    eNestState                              		:= E_NestState.IDLE;
    bSequenceToggle                         		:= FALSE; // Always restart from rotation step after reset
    GVL_MASTER.stNestTable.bNestStartCycle  		:= FALSE;
    GVL_MASTER.stNestTable.bNestInMotion    		:= FALSE;
    GVL_MASTER.stNestTable.qNestRotatePortA 		:= FALSE;
    GVL_MASTER.stNestTable.qNestRotatePortB 		:= FALSE;
    GVL_MASTER.stNestTable.bSupportExtendRequest    := FALSE;
    GVL_MASTER.stNestTable.bSupportRetractRequest   := TRUE;  // Safe home posture for elevator

    RETURN; // Abort remaining logic execution for this cycle
END_IF

// Global Safety Interlock: Force fault state immediately if air/safety is lost
IF NOT GVL_IO.stSafety.bSafetyOK AND GVL_Master.stMachineStatus.bFault THEN
    eNestState := E_NestState.FAULT;
END_IF

//eCurrentNestPos := M_GetCurrentPosition();

// =================================================================
// 2. INPUT SIGNAL PROCESSING (TRIGGERS)
// =================================================================
// Evaluate positive edge of the safety-certified two-hand control
rTrigTwoHands(CLK := GVL_IO.stSafety.bTwoHandsSafe);
tTwoHandTargetTime := REAL_TO_TIME(rHmiTwoHandPresetTime);   // Convert the HMI float milliseconds value into PLC TIME data type
tTwoHandHoldTimer(IN := GVL_IO.stSafety.bTwoHandsSafe, PT := tTwoHandTargetTime); // Execute the verification timer tied to the physical two-hand safety input

// Trigger processing to allow automated cycle start from IDLE state
// IF rTrigTwoHands.Q AND GVL_MASTER.bStations_Home AND GVL_IO.stSafety.bSafetyOK AND (eNestState = E_NestState.IDLE) THEN
//      IF GVL_MASTER.stMachineStatus.bAutoCycle THEN
//          GVL_MASTER.stNestTable.bNestInMotion := TRUE;
//          eNestState                           := E_NestState.ROTATING_TABLE; // Start the automated cycle directly at rotation step
//      END_IF
// END_IF

// =================================================================
// 3. TIMERS EXECUTION (CYCLIC COUPLING TO MAIN PROGRAM INSTANCES)
// =================================================================
// Enchained timers execution pattern to generate an automated timeline for the TESTING state
tRotatingTableDelay(IN  := (eNestState = E_NestState.ROTATING_TABLE), PT := T#500MS);
tPortB_ResetDelay(IN    := (eNestState = E_NestState.STOP_TABLE), PT := T#1S);

// TESTING TIMELINE: 
// 1. Initial 100ms settling delay starts when entering TESTING state
tSupportRetractDelay(IN := (eNestState = E_NestState.TESTING), PT := T#100MS);
// 2. 2-Second lift holding duration executes after the initial pause finishes
tSupportExtendDelay(IN  := (eNestState = E_NestState.TESTING) AND tSupportRetractDelay.Q, PT := T#200MS);

// Two-hand return timeout.
// If the operator does not press the two-hand control again within 1 second,
// the sequence goes to FAULT.
tTwoHandReturnTimeout(IN := (eNestState = E_NestState.WRONG_POSITION),PT := T#5S);

// =================================================================
// 4. NEST TABLE STATE MACHINE CONTROL (WITH INTERNAL INTERLOCKS)
// =================================================================
CASE GVL_Master.stMachineStatus.eMachineState OF    
    
    E_MachineState.SYSTEM_AUTO_CYCLE,
	E_MachineState.MANUAL_MODE:
        
        CASE eNestState OF
        
            E_NestState.IDLE:

				GVL_MASTER.stNestTable.qNestRotatePortA := FALSE;
				GVL_MASTER.stNestTable.qNestRotatePortB := FALSE;
				GVL_MASTER.stNestTable.bNestInMotion    := FALSE;
				GVL_MASTER.stProcess.bNestTestingReady  := FALSE;
			//
				IF GVL_IO.stSafety.bSafetyOK
				   AND rTrigTwoHands.Q
				   AND GVL_MASTER.bStations_Home
				   AND GVL_MASTER.stNestTable.bSupportRetracted
				   AND bNestSequenceAllowed
				   AND (
						GVL_MASTER.stMachineStatus.eMachineState =
							E_MachineState.MANUAL_MODE
						OR
						GVL_MASTER.stPuckLocker.bIndexPermissive
					)
				   AND stKistler_Status.bInPosition
				   AND NOT stKistler_Status.bBusy THEN
				
					GVL_MASTER.stNestTable.bNestInMotion := TRUE;
					eNestState := E_NestState.ROTATING_TABLE;
				
				END_IF
        
            E_NestState.ROTATING_TABLE: // State 2: ROTATING TABLE

				GVL_MASTER.stNestTable.bNestInMotion      := TRUE;
				GVL_MASTER.stProcess.bNestTestingReady    := FALSE;
				GVL_MASTER.stNestTable.bSupportExtendRequest := FALSE;
			    GVL_MASTER.stNestTable.bSupportRetractRequest := TRUE;
			
				IF NOT GVL_IO.stSafety.bSafetyOK THEN
			
					GVL_MASTER.stNestTable.qNestRotatePortA := FALSE;
					GVL_MASTER.stNestTable.qNestRotatePortB := FALSE;
					eNestState := E_NestState.FAULT;
			
				ELSIF NOT GVL_IO.stSafety.bTwoHandsSafe
					  AND NOT tTwoHandHoldTimer.Q THEN
			
					GVL_MASTER.stNestTable.qNestRotatePortA := FALSE;
					GVL_MASTER.stNestTable.qNestRotatePortB := FALSE;
					eNestState := E_NestState.WRONG_POSITION;
			
				ELSIF NOT bNestSequenceAllowed THEN
			
					GVL_MASTER.stNestTable.qNestRotatePortA := FALSE;
					GVL_MASTER.stNestTable.qNestRotatePortB := FALSE;
					eNestState := E_NestState.IDLE;
			
				ELSIF GVL_MASTER.stNestTable.bSupportRetracted 
					AND NOT stKistler_Status.bBusy 
					AND NOT GVL_MASTER.stActuators.bGuideCylinderExtendRequest
					AND stKistler_Status.bInPosition
					AND NOT GVL_MASTER.stProcess.bKistlerCycleRequest THEN
			
					GVL_MASTER.stNestTable.qNestRotatePortA := TRUE;
					GVL_MASTER.stNestTable.qNestRotatePortB := FALSE;
			
					IF tRotatingTableDelay.Q
					   AND GVL_MASTER.stNestTable.bNestCompletedSensor THEN
			
						eNestState := E_NestState.STOP_TABLE;
			
					END_IF
			
				ELSE
					// Support is not retracted. Do not rotate.
					GVL_MASTER.stNestTable.qNestRotatePortA := FALSE;
					GVL_MASTER.stNestTable.qNestRotatePortB := FALSE;
			
				END_IF
        
            E_NestState.STOP_TABLE: // State 3: STOP TABLE

				GVL_MASTER.stProcess.bNestTestingReady := FALSE;
			
				GVL_MASTER.stNestTable.qNestRotatePortA := FALSE;
				GVL_MASTER.stNestTable.qNestRotatePortB := TRUE;
			
				IF NOT GVL_IO.stSafety.bSafetyOK THEN
			
					GVL_MASTER.stNestTable.qNestRotatePortA := FALSE;
					GVL_MASTER.stNestTable.qNestRotatePortB := FALSE;
					eNestState := E_NestState.FAULT;
			
				ELSIF NOT bNestSequenceAllowed THEN
			
					GVL_MASTER.stNestTable.qNestRotatePortA := FALSE;
					GVL_MASTER.stNestTable.qNestRotatePortB := FALSE;
					GVL_MASTER.stNestTable.bNestInMotion    := FALSE;
					eNestState := E_NestState.IDLE;
			
				ELSIF tPortB_ResetDelay.Q
					  AND GVL_MASTER.stNestTable.bNestReadySensor
					  AND GVL_MASTER.stNestTable.bNestLockedSensor THEN
			
					GVL_MASTER.stNestTable.bNestInMotion    := FALSE;
					GVL_MASTER.stNestTable.qNestRotatePortB := FALSE;
					eNestState := E_NestState.TESTING;
			
				END_IF
        
			E_NestState.TESTING: // State 4: TESTING / Kistler test position
			
				GVL_MASTER.stNestTable.qNestRotatePortA := FALSE;
				GVL_MASTER.stNestTable.qNestRotatePortB := FALSE;
				GVL_MASTER.stNestTable.bNestInMotion := FALSE;
			
			
				IF NOT GVL_IO.stSafety.bSafetyOK THEN
			
					GVL_MASTER.stProcess.bNestTestingReady := FALSE;
					eNestState := E_NestState.FAULT;
			
			
				ELSIF NOT bNestSequenceAllowed THEN
			
					GVL_MASTER.stProcess.bNestTestingReady := FALSE;
					eNestState := E_NestState.IDLE;
			
			
				ELSIF NOT GVL_MASTER.stNestTable.bNestReadySensor
					  OR NOT GVL_MASTER.stNestTable.bNestLockedSensor
					  OR eCurrentNestPos = E_NestPosition.Unknown THEN
			
					GVL_MASTER.stProcess.bNestTestingReady := FALSE;
					eNestState := E_NestState.FAULT;
			
			
				ELSE
			
					// Table is stopped and safely positioned for the Kistler process.
					GVL_MASTER.stProcess.bNestTestingReady := TRUE;
			
			
					// The Process Cycle has completed the Kistler operation
					// and is requesting the nest to leave the testing phase.
					IF GVL_MASTER.stProcess.bReleaseNestRotation THEN
			
						GVL_MASTER.stProcess.bNestTestingReady := FALSE;
						GVL_MASTER.stProcess.bReleaseNestRotation := FALSE;
			
						// Do not rotate yet. First wait for the operator exchange.
						eNestState := E_NestState.WAIT_OPERATOR_EXCHANGE;
			
					END_IF
			
				END_IF
				
			E_NestState.WAIT_OPERATOR_EXCHANGE:

				// The Kistler test is finished.
				// Keep the table stationary while the operator completes:
				// - processed-part removal;
				// - puck exchange when required;
				// - new puck locking;
				// - new-part loading.
			
				GVL_MASTER.stNestTable.qNestRotatePortA := FALSE;
				GVL_MASTER.stNestTable.qNestRotatePortB := FALSE;
				GVL_MASTER.stNestTable.bNestInMotion 	:= FALSE;
			
				GVL_MASTER.stProcess.bNestTestingReady 		:= FALSE;
				GVL_MASTER.stProcess.bReleaseNestRotation 	:= FALSE;
			
			
				IF NOT GVL_IO.stSafety.bSafetyOK THEN
			
					eNestState := E_NestState.FAULT;
			
			
				ELSIF NOT bNestSequenceAllowed THEN
			
					eNestState := E_NestState.IDLE;
			
			
				ELSIF NOT GVL_MASTER.stNestTable.bNestReadySensor
					  OR NOT GVL_MASTER.stNestTable.bNestLockedSensor
					  OR eCurrentNestPos = E_NestPosition.Unknown THEN
			
					eNestState := E_NestState.FAULT;
			
			
				ELSIF     (
					GVL_MASTER.stMachineStatus.eMachineState =
						E_MachineState.MANUAL_MODE
					OR
					GVL_MASTER.stPuckLocker.bIndexPermissive
				) THEN
			
					// Operator exchange completed.
					// Return to IDLE, where the existing two-hand logic
					// can start the next pneumatic index.
					eNestState := E_NestState.IDLE;
			
				END_IF
			
				
				
			E_NestState.WRONG_POSITION: // State 99: WRONG_POSITION (Emergency Stop or Air Loss)

				GVL_MASTER.stNestTable.qNestRotatePortA := FALSE;
				GVL_MASTER.stNestTable.qNestRotatePortB := TRUE;
				GVL_MASTER.stNestTable.bNestInMotion    := TRUE;
			
				GVL_MASTER.stProcess.bNestTestingReady  := FALSE;
			
				IF tTwoHandReturnTimeout.Q THEN
			
					GVL_MASTER.stNestTable.qNestRotatePortA := FALSE;
					GVL_MASTER.stNestTable.qNestRotatePortB := FALSE;
					GVL_MASTER.stNestTable.bNestInMotion    := FALSE;
			
					eNestState := E_NestState.FAULT;
			
				ELSIF rTrigTwoHands.Q
					  AND GVL_IO.stSafety.bSafetyOK
					  AND bNestSequenceAllowed
					  AND GVL_MASTER.stNestTable.bSupportRetracted THEN
			
					GVL_MASTER.stNestTable.qNestRotatePortA := TRUE;
					GVL_MASTER.stNestTable.qNestRotatePortB := FALSE;
			
					eNestState := E_NestState.ROTATING_TABLE;
			
				ELSIF GVL_IO.stSafety.bSafetyOK
					  AND NOT GVL_MASTER.stMachineStatus.bFault
					  AND GVL_MASTER.stNestTable.bNestReadySensor
					  AND eCurrentNestPos <> E_NestPosition.Unknown THEN
			
					GVL_MASTER.stNestTable.qNestRotatePortA := FALSE;
					GVL_MASTER.stNestTable.qNestRotatePortB := FALSE;
					GVL_MASTER.stNestTable.bNestInMotion    := FALSE;
			
					eNestState := E_NestState.STOP_TABLE;
			
				END_IF
				
            E_NestState.FAULT:

					GVL_MASTER.stNestTable.qNestRotatePortA := FALSE;
					GVL_MASTER.stNestTable.qNestRotatePortB := FALSE;
					GVL_MASTER.stNestTable.bNestInMotion    := FALSE;
				
					GVL_MASTER.stProcess.bNestTestingReady  := FALSE;
					GVL_MASTER.stProcess.bReleaseNestRotation := FALSE;
				
					GVL_MASTER.stNestTable.bSupportExtendRequest  := FALSE;
					GVL_MASTER.stNestTable.bSupportRetractRequest := TRUE;
				
					GVL_MASTER.stMachineStatus.eMachineState := E_MachineState.FAULT;

        END_CASE

    // =================================================================
    // FAULT 
    // =================================================================
	
	E_MachineState.FAULT:
	
	 				GVL_MASTER.stNestTable.qNestRotatePortA := FALSE;
					GVL_MASTER.stNestTable.qNestRotatePortB := FALSE;
					GVL_MASTER.stNestTable.bNestInMotion    := FALSE;
				
					GVL_MASTER.stProcess.bNestTestingReady  := FALSE;
					GVL_MASTER.stProcess.bReleaseNestRotation := FALSE;
				
					GVL_MASTER.stNestTable.bSupportExtendRequest  := FALSE;
					GVL_MASTER.stNestTable.bSupportRetractRequest := TRUE;

	    IF GVL_IO.stSafety.bSafetyOK AND NOT GVL_Master.stMachineStatus.bFault THEN
        	eNestState := E_NestState.IDLE;
        END_IF

	

		
	END_CASE
END_METHOD

METHOD PRIVATE M_OperatorExchangeControl
VAR
	iOperatorNestIndex 	: INT;
    bOperatorResultPass : BOOL;
    bOperatorResultFail : BOOL;
	bOperatorResultValid : BOOL;
END_VAR
// Default value prevents stale index permission.
bOperatorExchangeComplete := FALSE;


// -----------------------------------------------------------------------------
// Validate the nest currently accessible to the operator.
// -----------------------------------------------------------------------------
IF eOperatorNestPosition = E_NestPosition.Unknown THEN
    RETURN;
END_IF


iOperatorNestIndex := TO_INT(eOperatorNestPosition);

IF (iOperatorNestIndex < 1) OR (iOperatorNestIndex > 4) THEN
    RETURN;
END_IF


// -----------------------------------------------------------------------------
// Result associated with the nest currently accessible to the operator.
// -----------------------------------------------------------------------------
bOperatorResultValid :=
    GVL_MASTER.astNestProcessResult[
        iOperatorNestIndex
    ].bResultValid;


bOperatorResultPass :=
    GVL_MASTER.astNestProcessResult[
        iOperatorNestIndex
    ].bResultValid
    AND
    GVL_MASTER.astNestProcessResult[
        iOperatorNestIndex
    ].bPass;


bOperatorResultFail :=
    GVL_MASTER.astNestProcessResult[
        iOperatorNestIndex
    ].bResultValid
    AND
    GVL_MASTER.astNestProcessResult[
        iOperatorNestIndex
    ].bFail;

// -----------------------------------------------------------------------------
// Retain operator actions even while the Kistler is processing another nest.
//
// Both the nest removal pulse and the reject sensor pulse last only one PLC
// scan. They must therefore be retained immediately and not only when the
// exchange state machine reaches the corresponding waiting state.
// -----------------------------------------------------------------------------

// A processed part was removed from the operator nest.
IF (
        bOperatorResultValid
        OR bPendingOperatorResultPass
        OR bPendingOperatorResultFail
   )
   AND GVL_MASTER.astNestTracking[
        iOperatorNestIndex
   ].bPartRemovedPulse THEN

    bPartRemovedConfirmedForExchange := TRUE;

END_IF


// A failed part was placed at the reject sensor.
IF (
        bOperatorResultFail
        OR bPendingOperatorResultFail
   )
   AND rtPartPresentReject.Q THEN

    bRejectConfirmedForExchange := TRUE;

END_IF


// ============================================================================
// Operator exchange sequence
// ============================================================================
CASE eOperatorExchangeState OF


    // ========================================================================
    E_OperatorExchangeState.Idle:
    // ========================================================================

        bOperatorExchangeComplete := FALSE;

        // Preserve the physical nest associated with this exchange.
        eCompletedOperatorExchangeNest :=
            eOperatorNestPosition;


        // --------------------------------------------------------------------
        // Case 1:
        // A tested result is pending at the operator nest.
        //
        // The processed part must be handled before the table may index.
        // --------------------------------------------------------------------
        IF
			(
				(
					eNestState = E_NestState.IDLE
					OR
					eNestState = E_NestState.WAIT_OPERATOR_EXCHANGE
					OR
					(
						eNestState = E_NestState.TESTING
						AND bOperatorResultPass
					)
				)
				AND NOT GVL_MASTER.stNestTable.bNestInMotion
				AND GVL_MASTER.stNestTable.bNestReadySensor
				AND GVL_MASTER.stNestTable.bNestLockedSensor
				AND bOperatorResultValid
			)
			THEN

            // Latch the result for the entire operator exchange.
            //
            // Do not reset these variables every PLC cycle.
            bPendingOperatorResultPass :=
                bOperatorResultPass;

            bPendingOperatorResultFail :=
                bOperatorResultFail;

           //bRejectConfirmedForExchange := FALSE;


			// -------------------------------------------------------------
			// The processed part may already have been removed while another
			// nest was being tested.
			//
			// If the operator already loaded a new part, the physical sensor
			// will be ON again. Therefore, the retained removal event must
			// take priority over the current sensor state.
			// -------------------------------------------------------------
			IF bPartRemovedConfirmedForExchange THEN
			
				// ---------------------------------------------------------
				// PASS result.
				// ---------------------------------------------------------
				IF bOperatorResultPass THEN
			
					IF GVL_HMI.stPuckLocker.eMode =
						E_PuckLockerMode.Disabled THEN
			
						eOperatorExchangeState :=
							E_OperatorExchangeState.ExchangeComplete;
			
					ELSE
			
						eOperatorExchangeState :=
							E_OperatorExchangeState.WaitingForPuckRemoval;
			
					END_IF
			
			
				// ---------------------------------------------------------
				// FAIL result.
				// ---------------------------------------------------------
				ELSIF bOperatorResultFail THEN
			
					eOperatorExchangeState :=
						E_OperatorExchangeState.WaitingForRejectConfirmation;
			
				END_IF
			
			
			// -------------------------------------------------------------
			// No removal event was retained and the processed part is still
			// physically present.
			//
			// Wait for the operator to remove it.
			// -------------------------------------------------------------
			ELSIF GVL_MASTER.stSensors.bPartPresent_NEST THEN
			
				eOperatorExchangeState :=
					E_OperatorExchangeState.WaitingForPartRemoval;
			
			
			// -------------------------------------------------------------
			// The part is already absent, for example after fault recovery
			// or machine restart.
			// -------------------------------------------------------------
			ELSE
			
				bPartRemovedConfirmedForExchange := TRUE;
			
				// ---------------------------------------------------------
				// PASS result.
				// ---------------------------------------------------------
				IF bOperatorResultPass THEN
			
					IF GVL_HMI.stPuckLocker.eMode =
						E_PuckLockerMode.Disabled THEN
			
						eOperatorExchangeState :=
							E_OperatorExchangeState.ExchangeComplete;
			
					ELSE
			
						eOperatorExchangeState :=
							E_OperatorExchangeState.WaitingForPuckRemoval;
			
					END_IF
			
			
				// ---------------------------------------------------------
				// FAIL result.
				// ---------------------------------------------------------
				ELSIF bOperatorResultFail THEN
			
					eOperatorExchangeState :=
						E_OperatorExchangeState.WaitingForRejectConfirmation;
			
				END_IF
			
			END_IF


        // --------------------------------------------------------------------
        // Case 2:
        // No tested result is pending.
        //
        // Enabled:
        //     Require a present and locked puck.
        //
        // Disabled:
        //     Ignore only the physical puck conditions.
        // --------------------------------------------------------------------
        ELSIF (
                eNestState = E_NestState.IDLE
                OR
                eNestState = E_NestState.WAIT_OPERATOR_EXCHANGE
              )
              AND NOT GVL_MASTER.stNestTable.bNestInMotion
              AND GVL_MASTER.stNestTable.bNestReadySensor
              AND GVL_MASTER.stNestTable.bNestLockedSensor
              AND NOT bOperatorResultValid
              AND (
                    GVL_HMI.stPuckLocker.eMode =
                        E_PuckLockerMode.Disabled

                    OR
                    (
                        GVL_MASTER.stPuckLocker.bPuckDetected
                        AND
                        GVL_MASTER.stPuckLocker.bPuckLocked
                        AND
                        GVL_MASTER.stPuckLocker.eState =
                            E_PuckLockerState.Locked
                    )
              ) THEN

            bPendingOperatorResultPass := FALSE;
            bPendingOperatorResultFail := FALSE;

            bPartRemovedConfirmedForExchange := FALSE;
            bRejectConfirmedForExchange := FALSE;

            eOperatorExchangeState :=
                E_OperatorExchangeState.ExchangeComplete;

        END_IF


    // ========================================================================
    E_OperatorExchangeState.WaitingForPartRemoval:
    // ========================================================================

        bOperatorExchangeComplete := FALSE;


        // This state is entered only when a processed part was confirmed
        // present in the operator nest.
        //
        // Therefore, the part has been removed when the physical sensor
        // becomes FALSE.
        IF bPartRemovedConfirmedForExchange
   			OR NOT GVL_MASTER.stSensors.bPartPresent_NEST THEN

            bPartRemovedConfirmedForExchange := TRUE;


            // -------------------------------------------------------------
            // PASS result.
            // -------------------------------------------------------------
            IF bPendingOperatorResultPass THEN

                // With the Puck Locker disabled, removal of the good part
                // completes the operator exchange.
                IF GVL_HMI.stPuckLocker.eMode =
                    E_PuckLockerMode.Disabled THEN

                    bPartRemovedConfirmedForExchange := FALSE;

                    eOperatorExchangeState :=
                        E_OperatorExchangeState.ExchangeComplete;

                ELSE

                    // Original enabled Puck Locker sequence.
                    eOperatorExchangeState :=
                        E_OperatorExchangeState.WaitingForPuckRemoval;

                END_IF


            // -------------------------------------------------------------
            // FAIL result.
            // -------------------------------------------------------------
            ELSIF bPendingOperatorResultFail THEN

                // The rejected part must be placed at the reject sensor.
                eOperatorExchangeState :=
                    E_OperatorExchangeState.WaitingForRejectConfirmation;

            END_IF

        END_IF


    // ========================================================================
    E_OperatorExchangeState.WaitingForPuckRemoval:
    // ========================================================================

        bOperatorExchangeComplete := FALSE;


        // Recovery protection:
        //
        // If the Puck Locker is disabled while the sequence is already in
        // this state, no puck removal must be awaited.
        IF GVL_HMI.stPuckLocker.eMode =
            E_PuckLockerMode.Disabled THEN

            bPartRemovedConfirmedForExchange := FALSE;

            eOperatorExchangeState :=
                E_OperatorExchangeState.ExchangeComplete;

        ELSE

            // Once the locker accepts the release request,
            // the part-removal handshake is no longer needed.
            IF GVL_MASTER.stPuckLocker.eState =
                E_PuckLockerState.ReleasingPuck THEN

                bPartRemovedConfirmedForExchange := FALSE;

            END_IF


            // Advance when the old puck is physically gone.
            //
            // Do not require the locker to remain in ReleasingPuck.
            IF NOT GVL_MASTER.stPuckLocker.bPuckDetected THEN

                eOperatorExchangeState :=
                    E_OperatorExchangeState.WaitingForNewPuck;

            END_IF

        END_IF


    // ========================================================================
    E_OperatorExchangeState.WaitingForRejectConfirmation:
    // ========================================================================

        bOperatorExchangeComplete := FALSE;


        // Latch the reject-bin sensor pulse.
        IF rtPartPresentReject.Q THEN

            bRejectConfirmedForExchange := TRUE;

        END_IF


        // Complete the rejected-part exchange when:
        //
        // 1. The rejected part has been confirmed at the reject sensor.
        // 2. The part is no longer present in the operator nest.
        // 3. The Puck Locker is disabled, or the puck remains present
        //    and locked.
        IF bRejectConfirmedForExchange
			   AND bPartRemovedConfirmedForExchange
			   AND
			   (
                GVL_HMI.stPuckLocker.eMode =
                    E_PuckLockerMode.Disabled

                OR
                (
                    GVL_MASTER.stPuckLocker.bPuckDetected
                    AND
                    GVL_MASTER.stPuckLocker.bPuckLocked
                    AND
                    GVL_MASTER.stPuckLocker.eState =
                        E_PuckLockerState.Locked
                )
           ) THEN

            bPartRemovedConfirmedForExchange := FALSE;

            eOperatorExchangeState :=
                E_OperatorExchangeState.ExchangeComplete;

        END_IF


    // ========================================================================
    E_OperatorExchangeState.WaitingForNewPuck:
    // ========================================================================

        bOperatorExchangeComplete := FALSE;


        // Recovery protection:
        //
        // A replacement puck is not required when the locker is disabled.
        IF GVL_HMI.stPuckLocker.eMode =
            E_PuckLockerMode.Disabled THEN

            eOperatorExchangeState :=
                E_OperatorExchangeState.ExchangeComplete;


        // Original enabled Puck Locker sequence.
        ELSIF GVL_MASTER.stPuckLocker.bPuckDetected THEN

            eOperatorExchangeState :=
                E_OperatorExchangeState.WaitingForPuckLocked;

        END_IF


    // ========================================================================
    E_OperatorExchangeState.WaitingForPuckLocked:
    // ========================================================================

        bOperatorExchangeComplete := FALSE;


        // Recovery protection:
        //
        // Physical puck locking is not required when the locker is disabled.
        IF GVL_HMI.stPuckLocker.eMode =
            E_PuckLockerMode.Disabled THEN

            eOperatorExchangeState :=
                E_OperatorExchangeState.ExchangeComplete;


        // Original enabled Puck Locker sequence.
        ELSIF GVL_MASTER.stPuckLocker.bPuckDetected
           AND GVL_MASTER.stPuckLocker.bPuckLocked
           AND GVL_MASTER.stPuckLocker.eState =
                E_PuckLockerState.Locked THEN

            // Loading a new part remains optional.
            eOperatorExchangeState :=
                E_OperatorExchangeState.ExchangeComplete;

        END_IF


    // ========================================================================
    E_OperatorExchangeState.WaitingForPartLoading:
    // ========================================================================

        // Original behavior preserved.
        //
        // Require an actual OFF -> ON transition from the operator nest
        // sensor. The puck must also be present and locked.
        IF GVL_MASTER.astNestTracking[
                iOperatorNestIndex
           ].bPartLoadedPulse
           AND GVL_MASTER.stPuckLocker.bPuckDetected
           AND GVL_MASTER.stPuckLocker.bPuckLocked
           AND GVL_MASTER.stPuckLocker.eState =
                E_PuckLockerState.Locked THEN

            eOperatorExchangeState :=
                E_OperatorExchangeState.ExchangeComplete;

        END_IF


    // ========================================================================
    E_OperatorExchangeState.ExchangeComplete:
    // ========================================================================

        // Keep the index permission active until the table starts moving.
        bOperatorExchangeComplete := TRUE;


        // The previous result and its disposition are complete.
        M_ClearCompletedOperatorNestResult();


        IF GVL_MASTER.stNestTable.bNestInMotion THEN

            bPendingOperatorResultPass := FALSE;
            bPendingOperatorResultFail := FALSE;

            bPartRemovedConfirmedForExchange := FALSE;
            bRejectConfirmedForExchange := FALSE;

            eOperatorExchangeState :=
                E_OperatorExchangeState.WaitingForTableIndexComplete;

        END_IF


    // ========================================================================
    E_OperatorExchangeState.WaitingForTableIndexComplete:
    // ========================================================================

        bOperatorExchangeComplete := TRUE;


        IF eNestState = E_NestState.TESTING
           AND NOT GVL_MASTER.stNestTable.bNestInMotion
           AND GVL_MASTER.stNestTable.bNestReadySensor
           AND GVL_MASTER.stNestTable.bNestLockedSensor
           AND eCurrentNestPos <> E_NestPosition.Unknown THEN

            bOperatorExchangeComplete := FALSE;

            bPendingOperatorResultPass := FALSE;
            bPendingOperatorResultFail := FALSE;

            bPartRemovedConfirmedForExchange := FALSE;
            bRejectConfirmedForExchange := FALSE;

            eOperatorExchangeState :=
                E_OperatorExchangeState.Idle;

        END_IF


    // ========================================================================
    ELSE
    // ========================================================================

        bOperatorExchangeComplete := FALSE;

        bPendingOperatorResultPass := FALSE;
        bPendingOperatorResultFail := FALSE;

        bPartRemovedConfirmedForExchange := FALSE;
        bRejectConfirmedForExchange := FALSE;

        eOperatorExchangeState :=
            E_OperatorExchangeState.Idle;

END_CASE
END_METHOD

METHOD PRIVATE M_PreExecution : BOOL
VAR

END_VAR
// =================================================================================
// SYSTEM TIMERS
// =================================================================================
// Update initialization and safety timers on every PLC scan cycle
tonSys_Init(IN := GVL_MASTER.stMachineStatus.bInitialising);
tonSys_InitTimeout(IN := GVL_MASTER.stMachineStatus.bInitialising);

// TwinSAFE circuit stabilization timer (10 seconds)
tonSafety(IN := (GVL_MASTER.stMachineStatus.eMachineState = E_MachineState.SAFETY), PT := T#10S);

// 
//  fbStopTrigger(CLK := GVL_Master.i_bButtonStop);
//  bButtonStop := fbStopTrigger.Q;

// =================================================================================
// HMI MESSAGE CLEARING
// =================================================================================
// Clear old system messages if the machine is not actively in production
// Uses the proper ENUM namespace from your MASTER folder
IF GVL_MASTER.stMachineStatus.eMachineState <> E_MachineState.SYSTEM_AUTO_CYCLE THEN
    sMachineMessage := '';            
END_IF


// =================================================================================
// CRITICAL FAULT INTERLOCK (Watchdog)
// =================================================================================
// If Kistler hardware is NOT ready, force the state machine to FAULT immediately
// Exception: Do not override if the system is currently in SAFETY or POWER_UP
IF NOT GVL_MASTER.bKistlerSystemReady 
    AND GVL_MASTER.stMachineStatus.eMachineState <> E_MachineState.SAFETY 
    AND GVL_MASTER.stMachineStatus.eMachineState <> E_MachineState.SYSTEM_POWER_UP THEN
    
    GVL_MASTER.stMachineStatus.eMachineState := E_MachineState.FAULT;
END_IF


// =================================================================================
// START LEDs BUTTON OFF
// =================================================================================
eMode_LED_Start := E_LEDs_Mode.OFF;
eMode_LED_Reset := E_LEDs_Mode.OFF;

// =================================================================================
// METHOD EXECUTION FEEDBACK (Return True)
// =================================================================================
// Returning TRUE confirms the pre-execution routine completed successfully
M_PreExecution := TRUE;
END_METHOD

METHOD M_ProcessCycle : BOOL
VAR
bControlledStopActive 	: BOOL;
rTrigTwoHands : R_TRIG; // Edge trigger to detect single press of the two-hand safety signal

bManualIndexerOnly        : BOOL;
bManualKistlerOnly        : BOOL;
bManualIndexerAndKistler  : BOOL;



END_VAR
// Process cycle is allowed during:
//
// 1. Automatic production.
// 2. Manual Mode when the Kistler or indexer manual function is enabled.
bProcessCycleAllowed :=
    (
        GVL_MASTER.stMachineStatus.eMachineState =
            E_MachineState.SYSTEM_AUTO_CYCLE
    )
    OR
    (
        GVL_MASTER.stMachineStatus.eMachineState =
            E_MachineState.MANUAL_MODE

        AND
        (
            GVL_HMI.i_bHMIKistlerManualEnable
            OR
            GVL_HMI.i_bHMIIndexerManualEnable
        )
    );


bManualIndexerOnly :=
    GVL_HMI.i_bHMIIndexerManualEnable
    AND NOT GVL_HMI.i_bHMIKistlerManualEnable;


bManualKistlerOnly :=
    GVL_HMI.i_bHMIKistlerManualEnable
    AND NOT GVL_HMI.i_bHMIIndexerManualEnable;


bManualIndexerAndKistler :=
    GVL_HMI.i_bHMIIndexerManualEnable
    AND GVL_HMI.i_bHMIKistlerManualEnable;


// -----------------------------------------------------------------------------
// If process execution is not permitted, reset the temporary process states.
//
// Stored nest PASS/FAIL results must not be cleared by M_ResetProcessCycle.
// -----------------------------------------------------------------------------
IF NOT bProcessCycleAllowed THEN

    M_ResetProcessCycle();

    RETURN;

END_IF


// -----------------------------------------------------------------------------
// Common timers and edge detections.
// -----------------------------------------------------------------------------
rTrigTwoHands(
    CLK := GVL_IO.stSafety.bTwoHandsSafe
);


tTwoHandTargetTime :=
    REAL_TO_TIME(rHmiTwoHandPresetTime);


tTwoHandHoldTimer(
    IN := GVL_IO.stSafety.bTwoHandsSafe,
    PT := tTwoHandTargetTime
);


rtPartPresentReject(
    CLK := GVL_MASTER.stSensors.bPartPresent_Reject
);


// ============================================================================
// COMMON POSITION AND TRACKING UPDATE
//
// These methods are required in both Auto and Manual Mode.
// ============================================================================
eCurrentNestPos :=
    M_GetCurrentPosition();


M_UpdateActiveNestPositions();

M_UpdateOperatorNestTracking();


// ============================================================================
// AUTOMATIC OPERATOR EXCHANGE
//
// The following methods belong only to automatic production.
//
// They must not:
//
// - send a PASS/FAIL disposition while in Manual Mode;
// - release a puck during Manual Mode;
// - clear a completed nest result during Manual Mode;
// - block manual index movement waiting for part removal;
// - block manual index movement waiting for reject confirmation;
// - block manual index movement waiting for a puck.
// ============================================================================
IF GVL_MASTER.stMachineStatus.eMachineState =
    E_MachineState.SYSTEM_AUTO_CYCLE THEN

    M_UpdatePuckLockerPartRemovalStatus();

    M_ConfirmPuckLockerDisposition();

    M_PuckLockerDisposition();

    M_OperatorExchangeControl();

ELSE

    // Prevent a stale removal confirmation from being sent to the
    // Puck Locker while the machine is operating manually.
    GVL_MASTER.stPuckLocker.bPartRemovedFromNest := FALSE;

END_IF


// -----------------------------------------------------------------------------
// Determine whether the current physical table position is different from
// the most recently processed Kistler position.
// -----------------------------------------------------------------------------
bNestNewPositionReady :=
    (
        eCurrentNestPos <> E_NestPosition.UNKNOWN
    )
    AND
    (
        eCurrentNestPos <> eLastTestedNestPos
    );


// -----------------------------------------------------------------------------
// Capture live Kistler values while an automatic or manual sequence is active.
//
// This does not store PASS/FAIL. It only updates the live maximum values.
// -----------------------------------------------------------------------------
IF GVL_MASTER.stProcess.bKistlerCycleRequest
   AND NOT stKistlerOutTelegram.bSequenceEnd THEN

    M_HMIKistlerResult(
        eNestPosition := eCurrentNestPos,
        bPartOK       := FALSE,
        bPartNOK      := FALSE,
        rForce        := stKistler_Status.rLiveForce,
        rDistance     := stKistler_Status.rLiveDistance,
        bResetValues  := FALSE
    );

END_IF


// ============================================================================
// PROCESS CYCLE COORDINATOR
// ============================================================================
CASE GVL_MASTER.stMachineStatus.eMachineState OF


    // ========================================================================
    // AUTOMATIC CYCLE
    // ========================================================================
    E_MachineState.SYSTEM_AUTO_CYCLE:

        CASE eProcessCycleState OF


            // =================================================================
            E_ProcessCycle_State.IDLE:
            // =================================================================

                GVL_MASTER.stProcess.bKistlerCycleRequest := FALSE;
                GVL_MASTER.stProcess.bKistlerCycleDone    := FALSE;
                GVL_MASTER.stProcess.bKistlerHomeDone     := FALSE;
                GVL_MASTER.stProcess.bReleaseNestRotation := FALSE;

                tonAfterKistlerDelay(IN := FALSE);

                IF bProcessCycleAllowed THEN

                    eProcessCycleState :=
                        E_ProcessCycle_State.WAIT_NEST_TESTING_READY;

                END_IF


            // =================================================================
            E_ProcessCycle_State.WAIT_NEST_TESTING_READY:
            // =================================================================

                GVL_MASTER.stProcess.bKistlerCycleRequest := FALSE;
                GVL_MASTER.stProcess.bReleaseNestRotation := FALSE;

                tonAfterKistlerDelay(IN := FALSE);


                IF NOT bProcessCycleAllowed THEN

                    eProcessCycleState :=
                        E_ProcessCycle_State.IDLE;


                // -------------------------------------------------------------
                // Invalid table position.
                //
                // Never execute the Kistler if the PLC cannot determine which
                // physical nest is currently at the test station.
                // -------------------------------------------------------------
                ELSIF GVL_MASTER.stProcess.bNestTestingReady
                      AND eNestState = E_NestState.TESTING
                      AND eCurrentNestPos =
                            E_NestPosition.UNKNOWN THEN

                    GVL_MASTER.stProcess.bKistlerCycleRequest := FALSE;
                    GVL_MASTER.stProcess.bReleaseNestRotation := FALSE;
                    GVL_MASTER.stProcess.bKistlerCycleDone    := FALSE;
                    GVL_MASTER.stProcess.bKistlerHomeDone     := FALSE;

                    eProcessCycleState :=
                        E_ProcessCycle_State.FAULT;


                // -------------------------------------------------------------
                // Same position already processed, or no part at Kistler.
                //
                // Do not execute another Kistler cycle. Release the table.
                // -------------------------------------------------------------
                ELSIF GVL_MASTER.stProcess.bNestTestingReady
                      AND eNestState = E_NestState.TESTING
                      AND GVL_MASTER.stNestTable.bNestReadySensor
                      AND GVL_MASTER.stNestTable.bNestLockedSensor
                      AND NOT GVL_MASTER.stNestTable.bNestInMotion
                      AND eCurrentNestPos <>
                            E_NestPosition.UNKNOWN
                      AND
                      (
                          NOT bNestNewPositionReady
                          OR
                          NOT GVL_MASTER.stSensors.bPartPresent_Kistler
                      ) THEN

                    GVL_MASTER.stProcess.bKistlerCycleRequest := FALSE;
                    GVL_MASTER.stProcess.bKistlerCycleDone    := FALSE;

                    // Kistler side is considered complete because there is
                    // no valid new part to test.
                    GVL_MASTER.stProcess.bKistlerHomeDone := TRUE;


                    IF bNestNewPositionReady THEN

                        // New position without a part.
                        // Remove any previous HMI measurement result.
                        M_HMIKistlerResult(
                            eNestPosition := eCurrentNestPos,
                            bPartOK       := FALSE,
                            bPartNOK      := FALSE,
                            rForce        := 0.0,
                            rDistance     := 0.0,
                            bResetValues  := TRUE
                        );

                        eLastTestedNestPos :=
                            eCurrentNestPos;

                    END_IF


                    GVL_MASTER.stProcess.bReleaseNestRotation := TRUE;

                    eProcessCycleState :=
                        E_ProcessCycle_State.RELEASE_NEST;


                // -------------------------------------------------------------
                // New enabled nest containing a part.
                //
                // Execute the Kistler sequence.
                // -------------------------------------------------------------
                ELSIF GVL_MASTER.stProcess.bNestTestingReady
                      AND eNestState = E_NestState.TESTING
                      AND GVL_MASTER.stNestTable.bNestReadySensor
                      AND GVL_MASTER.stNestTable.bNestLockedSensor
                      AND NOT GVL_MASTER.stNestTable.bNestInMotion
                      AND stKistler_Status.eKistlerState =
                            E_KistlerState.READY
                      AND NOT stKistler_Status.bError
                      AND NOT bKistlerRecoveryHomeRequest
                      AND bNestNewPositionReady
                      AND GVL_MASTER.stSensors.bPartPresent_Kistler
                      AND M_IsNestEnabled(eCurrentNestPos) THEN

                    GVL_MASTER.stProcess.bKistlerCycleDone := FALSE;
                    GVL_MASTER.stProcess.bKistlerHomeDone  := FALSE;

                    bKistlerResultStored := FALSE;


                    // Clear the previous HMI measurement values.
                    M_HMIKistlerResult(
                        eNestPosition := eCurrentNestPos,
                        bPartOK       := FALSE,
                        bPartNOK      := FALSE,
                        rForce        := 0.0,
                        rDistance     := 0.0,
                        bResetValues  := TRUE
                    );


                    eProcessCycleState :=
                        E_ProcessCycle_State.REQUEST_KISTLER;


                // -------------------------------------------------------------
                // Nest disabled from HMI.
                //
                // Skip the Kistler test and release the table normally.
                // -------------------------------------------------------------
                ELSIF GVL_MASTER.stProcess.bNestTestingReady
                      AND eNestState = E_NestState.TESTING
                      AND GVL_MASTER.stNestTable.bNestReadySensor
                      AND GVL_MASTER.stNestTable.bNestLockedSensor
                      AND NOT GVL_MASTER.stNestTable.bNestInMotion
                      AND eCurrentNestPos <>
                            E_NestPosition.UNKNOWN
                      AND bNestNewPositionReady
                      AND GVL_MASTER.stSensors.bPartPresent_Kistler
                      AND NOT M_IsNestEnabled(eCurrentNestPos) THEN

                    GVL_MASTER.stProcess.bKistlerCycleRequest := FALSE;
                    GVL_MASTER.stProcess.bKistlerCycleDone    := FALSE;
                    GVL_MASTER.stProcess.bKistlerHomeDone     := TRUE;


                    M_HMIKistlerResult(
                        eNestPosition := eCurrentNestPos,
                        bPartOK       := FALSE,
                        bPartNOK      := FALSE,
                        rForce        := 0.0,
                        rDistance     := 0.0,
                        bResetValues  := TRUE
                    );


                    eLastTestedNestPos :=
                        eCurrentNestPos;

                    GVL_MASTER.stProcess.bReleaseNestRotation :=
                        TRUE;

                    eProcessCycleState :=
                        E_ProcessCycle_State.RELEASE_NEST;

                END_IF


            // =================================================================
            E_ProcessCycle_State.REQUEST_KISTLER:
            // =================================================================

                GVL_MASTER.stProcess.bKistlerCycleRequest := TRUE;


                IF stKistler_Status.bError THEN

                    GVL_MASTER.stProcess.bKistlerCycleRequest :=
                        FALSE;

                    eProcessCycleState :=
                        E_ProcessCycle_State.FAULT;


                ELSIF stKistler_Status.eKistlerState <>
                      E_KistlerState.READY THEN

                    eProcessCycleState :=
                        E_ProcessCycle_State.WAIT_KISTLER_DONE;

                END_IF


            // =================================================================
            E_ProcessCycle_State.WAIT_KISTLER_DONE:
            // =================================================================

                // Keep the request active while the Kistler is executing.
                GVL_MASTER.stProcess.bKistlerCycleRequest := TRUE;


                IF stKistler_Status.bError THEN

                    GVL_MASTER.stProcess.bKistlerCycleRequest :=
                        FALSE;

                    eProcessCycleState :=
                        E_ProcessCycle_State.FAULT;


                ELSIF stKistler_Status.eKistlerState =
                      E_KistlerState.DONE THEN

                    GVL_MASTER.stProcess.bKistlerCycleRequest :=
                        FALSE;

                    GVL_MASTER.stProcess.bKistlerCycleDone :=
                        TRUE;

                    eProcessCycleState :=
                        E_ProcessCycle_State.WAIT_KISTLER_HOME;

                END_IF


            // =================================================================
            E_ProcessCycle_State.WAIT_KISTLER_HOME:
            // =================================================================

                M_StoreKistlerResult();

                GVL_MASTER.stProcess.bKistlerCycleRequest := FALSE;


                IF stKistler_Status.bError THEN

                    eProcessCycleState :=
                        E_ProcessCycle_State.FAULT;


                ELSIF stKistlerOutTelegram.bHomePosReached
                      OR stKistlerOutTelegram.bRefPosReached
                      OR stKistler_Status.bInPosition THEN

                    GVL_MASTER.test :=
                        GVL_MASTER.test + 1;

                    GVL_MASTER.stProcess.bKistlerHomeDone :=
                        TRUE;

                    GVL_MASTER.stProcess.bKistlerCycleDone :=
                        TRUE;


                    // ---------------------------------------------------------
                    // Store the process result.
                    // ---------------------------------------------------------
                    IF stKistler_Status.bPartOK THEN

                        GVL_MASTER.stProcess.bKistlerResultOK :=
                            TRUE;

                        GVL_MASTER.stProcess.bKistlerResultNOK :=
                            FALSE;


                    ELSIF stKistler_Status.bPartNOK THEN

                        GVL_MASTER.stProcess.bKistlerResultOK :=
                            FALSE;

                        GVL_MASTER.stProcess.bKistlerResultNOK :=
                            TRUE;


                    ELSE

                        // Test ended without a valid OK/NOK result.
                        // Preserve the existing behavior.
                        RETURN;

                    END_IF


                    eLastTestedNestPos :=
                        eCurrentNestPos;


                    IF NOT M_HMIKistlerResult(
                        eNestPosition := eCurrentNestPos,
                        bPartOK       := stKistler_Status.bPartOK,
                        bPartNOK      := stKistler_Status.bPartNOK,
                        rForce        := stKistler_Status.rLiveForce,
                        rDistance     := stKistler_Status.rLiveDistance,
                        bResetValues  := FALSE
                    ) THEN

                        RETURN;

                    END_IF


                    eProcessCycleState :=
                        E_ProcessCycle_State.WAIT_AFTER_KISTLER;

                END_IF


            // =================================================================
            E_ProcessCycle_State.WAIT_AFTER_KISTLER:
            // =================================================================

                IF stKistlerOutTelegram.bSequenceEnd
                   AND
                   (
                       stKistlerOutTelegram.bHomePosReached
                       OR
                       stKistlerOutTelegram.bRefPosReached
                       OR
                       stKistler_Status.bInPosition
                   ) THEN

                    GVL_MASTER.stProcess.bReleaseNestRotation :=
                        TRUE;

                    eProcessCycleState :=
                        E_ProcessCycle_State.RELEASE_NEST;

                END_IF


            // =================================================================
            E_ProcessCycle_State.RELEASE_NEST:
            // =================================================================

                // Keep the release request active until NestTableControl
                // consumes it.
                GVL_MASTER.stProcess.bReleaseNestRotation := TRUE;


                IF eNestState <> E_NestState.TESTING
                   OR NOT GVL_MASTER.stProcess.bNestTestingReady THEN

                    GVL_MASTER.stProcess.bReleaseNestRotation :=
                        FALSE;

                    GVL_MASTER.stProcess.bKistlerCycleRequest :=
                        FALSE;

                    GVL_MASTER.stProcess.bKistlerCycleDone :=
                        FALSE;

                    GVL_MASTER.stProcess.bKistlerHomeDone :=
                        FALSE;

                    tonAfterKistlerDelay(IN := FALSE);


                    eProcessCycleState :=
                        E_ProcessCycle_State.WAIT_NEST_TESTING_READY;

                END_IF


            // =================================================================
            E_ProcessCycle_State.FAULT:
            // =================================================================

                GVL_MASTER.stProcess.bKistlerCycleRequest := FALSE;
                GVL_MASTER.stProcess.bReleaseNestRotation := FALSE;

                tonAfterKistlerDelay(IN := FALSE);

                M_ResetProcessCycle();

                GVL_MASTER.stMachineStatus.eMachineState :=
                    E_MachineState.FAULT;


                IF GVL_MASTER.stMachineStatus.bStopped THEN

                    eProcessCycleState :=
                        E_ProcessCycle_State.IDLE;

                END_IF


            // =================================================================
            ELSE
            // =================================================================

                eProcessCycleState :=
                    E_ProcessCycle_State.IDLE;

        END_CASE


    // ========================================================================
    // MANUAL MODE
    // ========================================================================
    E_MachineState.MANUAL_MODE:

        CASE eProcessCycleState OF


            // =================================================================
            E_ProcessCycle_State.IDLE:
            // =================================================================

                GVL_MASTER.stProcess.bKistlerCycleRequest := FALSE;
                GVL_MASTER.stProcess.bKistlerCycleDone    := FALSE;
                GVL_MASTER.stProcess.bKistlerHomeDone     := FALSE;
                GVL_MASTER.stProcess.bReleaseNestRotation := FALSE;

                GVL_MASTER.stProcess.bKistlerResultOK  := FALSE;
                GVL_MASTER.stProcess.bKistlerResultNOK := FALSE;

                tonAfterKistlerDelay(IN := FALSE);


                IF bManualIndexerOnly
                   OR bManualIndexerAndKistler THEN

                    eProcessCycleState :=
                        E_ProcessCycle_State.WAIT_NEST_TESTING_READY;


                ELSIF bManualKistlerOnly
                      AND NOT GVL_MASTER.stProcess.bNestTestingReady
                      AND stKistler_Status.eKistlerState =
                            E_KistlerState.READY
                      AND NOT stKistler_Status.bError
                      AND NOT bKistlerRecoveryHomeRequest THEN

                    GVL_MASTER.stProcess.bNestTestingReady :=
                        FALSE;

                    eProcessCycleState :=
                        E_ProcessCycle_State.REQUEST_KISTLER;

                END_IF


            // =================================================================
            E_ProcessCycle_State.WAIT_NEST_TESTING_READY:
            // =================================================================

                GVL_MASTER.stProcess.bKistlerCycleRequest := FALSE;
                GVL_MASTER.stProcess.bReleaseNestRotation := FALSE;

                tonAfterKistlerDelay(IN := FALSE);


                IF NOT (
                    bManualIndexerOnly
                    OR bManualIndexerAndKistler
                ) THEN

                    eProcessCycleState :=
                        E_ProcessCycle_State.IDLE;


                ELSIF GVL_MASTER.stProcess.bNestTestingReady
                      AND eNestState = E_NestState.TESTING
                      AND bManualIndexerAndKistler
                      AND stKistler_Status.eKistlerState =
                            E_KistlerState.READY
                      AND NOT stKistler_Status.bError
                      AND NOT bKistlerRecoveryHomeRequest THEN

                    eProcessCycleState :=
                        E_ProcessCycle_State.REQUEST_KISTLER;


                ELSIF GVL_MASTER.stProcess.bNestTestingReady
                      AND eNestState = E_NestState.TESTING
                      AND bManualIndexerOnly THEN

                    GVL_MASTER.stProcess.bKistlerCycleRequest :=
                        FALSE;

                    GVL_MASTER.stProcess.bKistlerHomeDone :=
                        TRUE;

                    GVL_MASTER.stProcess.bReleaseNestRotation :=
                        TRUE;

                    eProcessCycleState :=
                        E_ProcessCycle_State.RELEASE_NEST;

                END_IF


            // =================================================================
            E_ProcessCycle_State.REQUEST_KISTLER:
            // =================================================================

                // Kistler already reacted.
                IF stKistler_Status.eKistlerState <>
                    E_KistlerState.READY THEN

                    eProcessCycleState :=
                        E_ProcessCycle_State.WAIT_KISTLER_DONE;


                // -------------------------------------------------------------
                // Manual Kistler only.
                //
                // Start only on the two-hand rising edge.
                // -------------------------------------------------------------
                ELSIF bManualKistlerOnly
                      AND GVL_IO.stSafety.bSafetyOK
                      AND rTrigTwoHands.Q
                      AND GVL_MASTER.stNestTable.bNestReadySensor
                      AND GVL_MASTER.stNestTable.bNestLockedSensor
                      AND NOT stKistler_Status.bError
                      AND NOT bKistlerRecoveryHomeRequest THEN

                    GVL_MASTER.stProcess.bKistlerCycleRequest :=
                        TRUE;


                // -------------------------------------------------------------
                // Manual indexer and Kistler.
                // -------------------------------------------------------------
                ELSIF bManualIndexerAndKistler
                      AND GVL_MASTER.stProcess.bNestTestingReady
                      AND eNestState = E_NestState.TESTING
                      AND GVL_MASTER.stNestTable.bNestReadySensor
                      AND GVL_MASTER.stNestTable.bNestLockedSensor
                      AND NOT GVL_MASTER.stNestTable.bNestInMotion
                      AND eCurrentNestPos <>
                            E_NestPosition.UNKNOWN
                      AND bNestNewPositionReady
                      AND NOT stKistler_Status.bError
                      AND NOT bKistlerRecoveryHomeRequest THEN

                    GVL_MASTER.stProcess.bKistlerCycleRequest :=
                        TRUE;


                ELSIF stKistler_Status.bError THEN

                    GVL_MASTER.stProcess.bKistlerCycleRequest :=
                        FALSE;

                    eProcessCycleState :=
                        E_ProcessCycle_State.FAULT;

                END_IF


            // =================================================================
            E_ProcessCycle_State.WAIT_KISTLER_DONE:
            // =================================================================

                GVL_MASTER.stProcess.bKistlerCycleRequest := TRUE;


                IF stKistler_Status.bError THEN

                    GVL_MASTER.stProcess.bKistlerCycleRequest :=
                        FALSE;

                    eProcessCycleState :=
                        E_ProcessCycle_State.FAULT;


                ELSIF stKistler_Status.eKistlerState =
                      E_KistlerState.DONE THEN

                    // Capture the final available measurements.
                    M_HMIKistlerResult(
                        eNestPosition := eCurrentNestPos,
                        bPartOK       := FALSE,
                        bPartNOK      := FALSE,
                        rForce        := stKistler_Status.rLiveForce,
                        rDistance     := stKistler_Status.rLiveDistance,
                        bResetValues  := FALSE
                    );


                    GVL_MASTER.stProcess.bKistlerCycleRequest :=
                        FALSE;

                    GVL_MASTER.stProcess.bKistlerCycleDone :=
                        TRUE;


                    IF bManualIndexerAndKistler THEN

                        eLastTestedNestPos :=
                            eCurrentNestPos;

                        eProcessCycleState :=
                            E_ProcessCycle_State.WAIT_KISTLER_HOME;

                    ELSE

                        eProcessCycleState :=
                            E_ProcessCycle_State.IDLE;

                    END_IF

                END_IF


            // =================================================================
            E_ProcessCycle_State.WAIT_KISTLER_HOME:
            // =================================================================

                GVL_MASTER.stProcess.bKistlerCycleRequest := FALSE;


                IF stKistler_Status.bError THEN

                    eProcessCycleState :=
                        E_ProcessCycle_State.FAULT;


                ELSIF stKistlerOutTelegram.bHomePosReached
                      OR stKistlerOutTelegram.bRefPosReached
                      OR stKistler_Status.bInPosition THEN

                    GVL_MASTER.stProcess.bKistlerHomeDone :=
                        TRUE;


                    IF bManualIndexerAndKistler THEN

                        eProcessCycleState :=
                            E_ProcessCycle_State.WAIT_AFTER_KISTLER;

                    ELSE

                        eProcessCycleState :=
                            E_ProcessCycle_State.IDLE;

                    END_IF

                END_IF


            // =================================================================
            E_ProcessCycle_State.WAIT_AFTER_KISTLER:
            // =================================================================

                IF stKistlerOutTelegram.bSequenceEnd
                   AND
                   (
                       stKistlerOutTelegram.bHomePosReached
                       OR
                       stKistlerOutTelegram.bRefPosReached
                       OR
                       stKistler_Status.bInPosition
                   ) THEN

                    GVL_MASTER.stProcess.bReleaseNestRotation :=
                        TRUE;

                    eProcessCycleState :=
                        E_ProcessCycle_State.RELEASE_NEST;

                END_IF


            // =================================================================
            E_ProcessCycle_State.RELEASE_NEST:
            // =================================================================

                GVL_MASTER.stProcess.bReleaseNestRotation :=
                    TRUE;


                IF eNestState <> E_NestState.TESTING
                   OR NOT GVL_MASTER.stProcess.bNestTestingReady THEN

                    GVL_MASTER.stProcess.bReleaseNestRotation :=
                        FALSE;

                    GVL_MASTER.stProcess.bKistlerCycleRequest :=
                        FALSE;

                    GVL_MASTER.stProcess.bKistlerCycleDone :=
                        FALSE;

                    GVL_MASTER.stProcess.bKistlerHomeDone :=
                        FALSE;

                    tonAfterKistlerDelay(IN := FALSE);


                    IF bManualIndexerOnly
                       OR bManualIndexerAndKistler THEN

                        eProcessCycleState :=
                            E_ProcessCycle_State.WAIT_NEST_TESTING_READY;

                    ELSE

                        eProcessCycleState :=
                            E_ProcessCycle_State.IDLE;

                    END_IF

                END_IF


            // =================================================================
            E_ProcessCycle_State.FAULT:
            // =================================================================

                GVL_MASTER.stProcess.bKistlerCycleRequest :=
                    FALSE;

                GVL_MASTER.stProcess.bReleaseNestRotation :=
                    FALSE;

                tonAfterKistlerDelay(IN := FALSE);

                M_ResetProcessCycle();

                GVL_MASTER.stMachineStatus.eMachineState :=
                    E_MachineState.FAULT;


            // =================================================================
            ELSE
            // =================================================================

                eProcessCycleState :=
                    E_ProcessCycle_State.IDLE;

        END_CASE


    // ========================================================================
    ELSE
    // ========================================================================

        // This should normally be handled by bProcessCycleAllowed at the
        // beginning of the method.
        M_ResetProcessCycle();

END_CASE


M_ProcessCycle := TRUE;
END_METHOD

METHOD PRIVATE M_PuckLockerDisposition
VAR
	iOperatorNestIndex : INT;
    bResultPass        : BOOL;
    bResultFail        : BOOL;
END_VAR
// -----------------------------------------------------------------------------
// The operator nest must be known.
// -----------------------------------------------------------------------------
IF eOperatorNestPosition = E_NestPosition.Unknown THEN
    RETURN;
END_IF


// Process the operator disposition whenever the table is stationary,
// mechanically locked and accessible to the operator.
//
// TESTING:
//     Normal production flow.
//
// WAIT_OPERATOR_EXCHANGE:
//     Normal exchange after a completed test.
//
// IDLE:
//     Recovery flow after FAULT, STOPPED or reinitialisation.
IF (
        eNestState <> E_NestState.IDLE
        AND eNestState <> E_NestState.TESTING
        AND eNestState <> E_NestState.WAIT_OPERATOR_EXCHANGE
   )
   OR GVL_MASTER.stNestTable.bNestInMotion
   OR NOT GVL_MASTER.stNestTable.bNestReadySensor
   OR NOT GVL_MASTER.stNestTable.bNestLockedSensor
   OR eCurrentNestPos = E_NestPosition.Unknown THEN

    RETURN;

END_IF


// -----------------------------------------------------------------------------
// E_NestPosition values correspond directly to array indexes 1..4.
// -----------------------------------------------------------------------------
iOperatorNestIndex := TO_INT(eOperatorNestPosition);

IF (iOperatorNestIndex < 1) OR (iOperatorNestIndex > 4) THEN
    RETURN;
END_IF


// -----------------------------------------------------------------------------
// The nest currently accessible to the operator must contain a valid result.
// -----------------------------------------------------------------------------
IF NOT GVL_MASTER.astNestProcessResult[iOperatorNestIndex].bResultValid THEN
    RETURN;
END_IF


// -----------------------------------------------------------------------------
// Do not process the same nest disposition more than once.
// -----------------------------------------------------------------------------
IF GVL_MASTER.astNestProcessResult[iOperatorNestIndex].bDispositionSent THEN
    RETURN;
END_IF


// -----------------------------------------------------------------------------
// Copy the result locally for validation and readability.
// -----------------------------------------------------------------------------
bResultPass :=
    GVL_MASTER.astNestProcessResult[iOperatorNestIndex].bPass;

bResultFail :=
    GVL_MASTER.astNestProcessResult[iOperatorNestIndex].bFail;


// -----------------------------------------------------------------------------
// The result must contain exactly one disposition.
//
// Invalid combinations:
//     PASS = FALSE and FAIL = FALSE
//     PASS = TRUE  and FAIL = TRUE
// -----------------------------------------------------------------------------
IF bResultPass = bResultFail THEN
    RETURN;
END_IF


// -----------------------------------------------------------------------------
// PUCK LOCKER DISABLED:
//
// There is no physical locker handshake to perform.
//
// Mark the disposition as delivered internally so that the operator exchange
// sequence can continue using the normal PASS/FAIL result.
//
// FAIL still requires:
//     1. Part removal from the operator nest.
//     2. Confirmation from the reject-bin sensor.
//
// No puck presence or puck locked condition is required.
// -----------------------------------------------------------------------------
IF GVL_HMI.stPuckLocker.eMode = E_PuckLockerMode.Disabled THEN

    GVL_MASTER.astNestProcessResult[
        iOperatorNestIndex
    ].bDispositionSent := TRUE;

    RETURN;

END_IF


// -----------------------------------------------------------------------------
// A previous disposition was already sent and is still waiting for confirmation
// from PRG_PuckLocker.
// -----------------------------------------------------------------------------
IF ePendingPuckDispositionNest <> E_NestPosition.Unknown THEN
    RETURN;
END_IF


// -----------------------------------------------------------------------------
// Do not overwrite a disposition that has not yet been consumed by the locker.
// -----------------------------------------------------------------------------
IF GVL_MASTER.stPuckLocker.bApplyDisposition
   OR GVL_MASTER.stPuckLocker.bDispositionPending THEN

    RETURN;

END_IF


// -----------------------------------------------------------------------------
// PASS:
// Authorise the release of one puck.
// -----------------------------------------------------------------------------
IF bResultPass THEN

    GVL_MASTER.stPuckLocker.nRequestedRelease := 1;
    GVL_MASTER.stPuckLocker.nRequestedRemoval := 0;

    // Store the nest that originated this request so that the confirmation
    // remains associated with the correct nest even if the table moves later.
    ePendingPuckDispositionNest :=
        eOperatorNestPosition;

    // Apply the request only after all associated data has been prepared.
    GVL_MASTER.stPuckLocker.bApplyDisposition := TRUE;


// -----------------------------------------------------------------------------
// FAIL:
// Inform the locker of the rejected result, but do not authorise puck release.
// The puck must remain locked until a future PASS result is received.
// -----------------------------------------------------------------------------
ELSIF bResultFail THEN

    GVL_MASTER.stPuckLocker.nRequestedRelease := 0;
    GVL_MASTER.stPuckLocker.nRequestedRemoval := 1;

    ePendingPuckDispositionNest :=
        eOperatorNestPosition;

    // Apply the request only after all associated data has been prepared.
    GVL_MASTER.stPuckLocker.bApplyDisposition := TRUE;

END_IF
END_METHOD

METHOD PRIVATE M_ResetProcessCycle : BOOL
VAR_INPUT

END_VAR

M_ResetProcessCycle := FALSE;

eProcessCycleState := E_ProcessCycle_State.IDLE;


// =========================================================
// RESET PROCESS FLAGS
// =========================================================

GVL_MASTER.stProcess.bKistlerCycleRequest := FALSE;
GVL_MASTER.stProcess.bKistlerCycleDone := FALSE;
GVL_MASTER.stProcess.bKistlerHomeDone := FALSE;
GVL_MASTER.stProcess.bNestTestingReady := FALSE;
GVL_MASTER.stProcess.bReleaseNestRotation := FALSE;
GVL_MASTER.stProcess.bKistlerResultOK := FALSE;
GVL_MASTER.stProcess.bKistlerResultNOK := FALSE;


// =========================================================
// RESET PROCESS TIMERS
// =========================================================

tonGuideCylinderDelay(IN := FALSE);
tonGuideCylinderRetractDelay(IN := FALSE);
tonAfterKistlerDelay(IN := FALSE);


// =========================================================
// RESET ACTUATOR REQUESTS
// =========================================================

GVL_MASTER.stActuators.bGuideCylinderExtendRequest := FALSE;

GVL_MASTER.stNestTable.bSupportExtendRequest := FALSE;
GVL_MASTER.stNestTable.bSupportRetractRequest := TRUE;


// =========================================================
// RESET HMI MANUAL COMMANDS
// =========================================================

GVL_HMI.i_bHMIManualModeRequest := FALSE;
GVL_HMI.i_bHMIIndexerManualEnable := FALSE;
GVL_HMI.i_bHMIKistlerManualEnable := FALSE;


// =========================================================
// RESET KISTLER SEQUENCE COMMANDS
// =========================================================

stKistler_CMD.bStart := FALSE;
stKistler_CMD.bRunSequence := FALSE;
stKistler_CMD.bDriveToHome := FALSE;
stKistler_CMD.bDriveToRef := FALSE;
stKistler_CMD.bContinueFromWait := FALSE;
stKistler_CMD.bTareY := FALSE;


// =========================================================
// START RESET PULSE
// =========================================================

// Start the pulse only on the first execution
IF NOT bKistlerResetPulse AND NOT tonKistlerReset.Q THEN
    bKistlerResetPulse := TRUE;
END_IF;


// Reset/Acknowledge command sent to the Kistler
stKistler_CMD.bReset := bKistlerResetPulse;


// Do not send Abort at the same time as Reset
stKistler_CMD.bAbort := NOT bKistlerResetPulse;


// =========================================================
// RESET PULSE TIMER
// =========================================================

tonKistlerReset(
    IN := bKistlerResetPulse,
    PT := T#500MS
);


// =========================================================
// RESET ROUTINE COMPLETE
// =========================================================

IF tonKistlerReset.Q THEN

    // End pulse commands
    bKistlerResetPulse := FALSE;

    stKistler_CMD.bReset := FALSE;
    stKistler_CMD.bAbort := FALSE;

    // Reset the timer for the next fault/reset
    tonKistlerReset(IN := FALSE);

    // Request recovery movement on the next initialization
    bKistlerRecoveryHomeRequest := TRUE;

    // Inform caller that the reset routine is complete
    M_ResetProcessCycle := TRUE;

END_IF;
END_METHOD

METHOD PRIVATE M_StatusMapping : BOOL
VAR_INPUT



END_VAR

// =================================================================================
// KISTLER TO GLOBAL STATUS MAPPING
// =================================================================================
// Link the software/hardware safety loop to the machine status structure
GVL_MASTER.stMachineStatus.bSafety := GVL_IO.stSafety.bSystemSafeOK;

// Map the local Kistler hardware ready flag to our main control variable
bKistlerReady := stKistler_Status.bReady;

// Update the global machine fault status if the Kistler press enters an error state
IF stKistler_Status.bError THEN
	GVL_MASTER.stMachineStatus.bFault := TRUE;
END_IF

// =================================================================================
// HMI / PANEL LAMP SIGNALLING MANAGEMENT
// =================================================================================
// Control the Start Button Lamp feedback based on machine state
IF GVL_MASTER.stMachineStatus.eMachineState = E_MachineState.STOPPED AND bKistlerReady THEN
    GVL_MASTER.bStartButtonLamp := GVL_MASTER.bBlink_1Hz; // Uses standard 1Hz global clock bit
ELSIF GVL_MASTER.stMachineStatus.eMachineState = E_MachineState.SYSTEM_AUTO_CYCLE THEN
    GVL_MASTER.bStartButtonLamp := TRUE;
ELSE
    GVL_MASTER.bStartButtonLamp := FALSE;
END_IF
// =================================================================================
// METHOD EXECUTION FEEDBACK (Return True)
// =================================================================================
// Returning TRUE confirms that the status mapping routine executed successfully
M_StatusMapping := TRUE;
END_METHOD

METHOD M_StoreKistlerResult
VAR
	iNestIndex : INT;
END_VAR
IF eKistlerNestPosition = E_NestPosition.Unknown THEN
    RETURN;
END_IF;

iNestIndex := eKistlerNestPosition;

IF (iNestIndex < 1) OR (iNestIndex > 4) THEN
    RETURN;
END_IF;

// Prevent writing the same result repeatedly for several PLC scans.
IF bKistlerResultStored THEN
    RETURN;
END_IF;

IF stKistler_Status.bPartOK THEN

    GVL_MASTER.astNestProcessResult[iNestIndex].bResultValid := TRUE;
    GVL_MASTER.astNestProcessResult[iNestIndex].bPass := TRUE;
    GVL_MASTER.astNestProcessResult[iNestIndex].bFail := FALSE;
    GVL_MASTER.astNestProcessResult[iNestIndex].bDispositionSent := FALSE;

    bKistlerResultStored := TRUE;

ELSIF stKistler_Status.bPartNOK THEN

    GVL_MASTER.astNestProcessResult[iNestIndex].bResultValid := TRUE;
    GVL_MASTER.astNestProcessResult[iNestIndex].bPass := FALSE;
    GVL_MASTER.astNestProcessResult[iNestIndex].bFail := TRUE;
    GVL_MASTER.astNestProcessResult[iNestIndex].bDispositionSent := FALSE;

    bKistlerResultStored := TRUE;

END_IF;
END_METHOD

METHOD M_SupportControl
VAR_INPUT
    bExtendRequest  : BOOL; // Request to lift support
    bRetractRequest : BOOL; // Request to lower support
END_VAR
// =================================================================
// SUPPORT CYLINDER CONTROL
// =================================================================
// This method is responsible only for the support cylinder outputs.
// It does not decide Auto Cycle or Manual Mode.
// The request must come from M_ProcessCycle, M_NestTableControl,
// or later from the Kistler coordination logic.

// Safety priority: never command both coils at the same time.
IF bExtendRequest AND NOT bRetractRequest THEN

    // Lift support
    GVL_MASTER.stNestTable.qSupportExtend  := TRUE;
    GVL_MASTER.stNestTable.qSupportRetract := FALSE;


ELSIF bRetractRequest AND NOT bExtendRequest THEN

    // Lower support
    GVL_MASTER.stNestTable.qSupportExtend  := FALSE;
    GVL_MASTER.stNestTable.qSupportRetract := TRUE;



ELSE

    // No request or conflicting request:
    // keep both outputs off to avoid fighting the pneumatic valve.
    GVL_MASTER.stNestTable.qSupportExtend  := FALSE;
    GVL_MASTER.stNestTable.qSupportRetract := FALSE;



END_IF
END_METHOD

METHOD PRIVATE M_UpdateActiveNestPositions
VAR_INPUT
END_VAR
eKistlerNestPosition := eCurrentNestPos;

eOperatorNestPosition := F_GetOppositeNestPosition( eKistlerPosition := eKistlerNestPosition );

IF eKistlerNestPosition <> E_NestPosition.Unknown THEN

    iKistlerNestIndex := TO_INT(eKistlerNestPosition);

ELSE

    iKistlerNestIndex := 0;

END_IF;

IF eOperatorNestPosition <> E_NestPosition.Unknown THEN

    iOperatorNestIndex := TO_INT(eOperatorNestPosition);

ELSE

    iOperatorNestIndex := 0;

END_IF;
END_METHOD

METHOD PRIVATE M_UpdateOperatorInstruction
VAR_INPUT
END_VAR
END_METHOD

METHOD PRIVATE M_UpdateOperatorNestTracking
VAR
	iOperatorNestIndex 	: INT;
    iNest               : INT;
    bPartPresent        : BOOL;
END_VAR
// Pulses are valid for one PLC scan only.
// Clear all previous events before evaluating the current operator nest.
FOR iNest := 1 TO 4 DO

    GVL_MASTER.astNestTracking[iNest].bPartRemovedPulse := FALSE;
    GVL_MASTER.astNestTracking[iNest].bPartLoadedPulse := FALSE;

END_FOR

// Track the operator sensor while the table is safely stationary.
// IDLE is required for the initial loading sequence.
// TESTING is required for the normal unload/reload sequence.
IF (
        eNestState <> E_NestState.IDLE
        AND eNestState <> E_NestState.TESTING
        AND eNestState <> E_NestState.WAIT_OPERATOR_EXCHANGE
   )
   OR GVL_MASTER.stNestTable.bNestInMotion
   OR NOT GVL_MASTER.stNestTable.bNestReadySensor
   OR NOT GVL_MASTER.stNestTable.bNestLockedSensor
   OR eOperatorNestPosition = E_NestPosition.Unknown THEN

    RETURN;

END_IF

// E_NestPosition corresponds to indexes 1..4.
iOperatorNestIndex := TO_INT(eOperatorNestPosition);

IF (iOperatorNestIndex < 1) OR (iOperatorNestIndex > 4) THEN
    RETURN;
END_IF

// The physical sensor represents the nest currently accessible
// to the operator.
bPartPresent := GVL_MASTER.stSensors.bPartPresent_NEST;

// Detect processed part removal.
GVL_MASTER.astNestTracking[iOperatorNestIndex].bPartRemovedPulse := GVL_MASTER.astNestTracking[iOperatorNestIndex].bPreviousSensor AND NOT bPartPresent;

// Detect new part loading.
GVL_MASTER.astNestTracking[iOperatorNestIndex].bPartLoadedPulse := NOT GVL_MASTER.astNestTracking[iOperatorNestIndex].bPreviousSensor AND bPartPresent;

// Store the current occupancy status.
GVL_MASTER.astNestTracking[iOperatorNestIndex].bPartLoaded := bPartPresent;

// Save the current sensor state for the next scan.
GVL_MASTER.astNestTracking[iOperatorNestIndex].bPreviousSensor := bPartPresent;
END_METHOD

METHOD PRIVATE M_UpdatePuckLockerPartRemovalStatus
VAR
	iOperatorNestIndex : INT;
END_VAR
// Keep the removal confirmation active until the Puck Locker
// acknowledges it by leaving the Locked state.
//
// Do not forward the one-scan physical sensor pulse directly.
GVL_MASTER.stPuckLocker.bPartRemovedFromNest := bPendingOperatorResultPass AND bPartRemovedConfirmedForExchange;
END_METHOD

METHOD PRIVATE M_UpdatePuckLockerPermissives
VAR_INPUT
END_VAR
// Puck Locker is considered permissive when disabled,
// or when enabled without any latched locker fault.
GVL_MASTER.stPuckLocker.bMachinePermissive :=
    (GVL_HMI.stPuckLocker.eMode = E_PuckLockerMode.Disabled)
    OR (
        NOT GVL_MASTER.stPuckLocker.bUnexpectedRemovalFault
        AND NOT GVL_MASTER.stPuckLocker.bPuckSensorMismatch
        AND GVL_MASTER.stPuckLocker.eState <>
            E_PuckLockerState.UnexpectedPuckRemovalFault
    );


// Index movement always depends on completion of the operator exchange.
//
// When the Puck Locker is disabled, its physical sensors and locker faults
// are bypassed through bMachinePermissive, but the operator must still:
//
//     1. Remove the processed part from the nest.
//     2. Place a failed part in the reject sensor.
//     3. Complete the operator exchange sequence.
//
// The Unknown-position exception is retained for initialisation/recovery.
GVL_MASTER.stPuckLocker.bIndexPermissive :=
    GVL_MASTER.stPuckLocker.bMachinePermissive
    AND (
        bOperatorExchangeComplete
        OR eCurrentNestPos = E_NestPosition.Unknown
    );
END_METHOD

END_PROGRAM

// ---- POUs/02_HMI/PGR_HMI.TcPOU
PROGRAM PGR_HMI
VAR
    // =========================================================================
    // SYSTEM & SYSTEM TIME MANAGEMENT
    // =========================================================================
    fbLocalTime         : FB_LocalSystemTime; // Fetches the local NT system time
    sTimeReal           : STRING;             // Formatted real-time string (HH:MM:SS)
    sDateReal           : STRING;             // Formatted real-date string (YYYY-MM-DD)
    sCurrentTimeStr     : STRING;             // General purpose timestamp string

    // =========================================================================
    // HMI BLINK & VISUAL FLASHING LOGIC
    // =========================================================================
    bFlash              : BOOL;               // Toggling bit for HMI flashing elements
    fbBlinkTimer        : TON;                // Timer driving the flashing pulse
    bBlinkTimer_Q_Old   : BOOL;               // Edge detection auxiliary bit for the timer

    // =========================================================================
    // IPC POWER CONTROL (REBOOT & SHUTDOWN)
    // =========================================================================
   // ePowerCmd           : E_PLC_Power := E_PLC_Power.Idle; // Command received from HMI
    fbReboot            : NT_Reboot;          // Operating system reboot execution block
    fbShutdown          : NT_Shutdown;        // Operating system shutdown execution block
	fbKillEdge 			: NT_StartProcess;    // close HMI
    tonRebootDelay      : TON;                // 30-second delay timer before rebooting
    bTriggerReboot      : BOOL;               // Internal trigger for fbReboot
    bTriggerShutdown    : BOOL;               // Internal trigger for fbShutdown
	bTriggerExitHMI     : BOOL;               // Internal trigger for fbShutdown
	bErrorOut : BOOL;
	nErrIDOut : UDINT;
	tonPowerDelay       : TON;     // Timer unificado de 60 segundos para Reboot/Shutdown
	iCountdownValue     : INT;     // Valor regressivo (60 a 0) enviado para a IHM
	

    // =========================================================================
    // TESTING & ALARM SIMULATION
    // =========================================================================
    bTriggerTestAlarm   : BOOL;               // Force TRUE online to simulate a HMI alarm
    fbTestAlarmTrigger  : R_TRIG;             // Rising edge detector for the test alarm
    bResetTest          : BOOL;               // Reset command for test sequences

    // =========================================================================
    // BUFFER / TABLE ARRAYS INDEXES
    // =========================================================================
    i                   : DINT;               // Generic loop index iterator
    n                   : DINT;               // Specific table data index pointer
END_VAR

// =================================================================
// RUN GENERATOR CLOCK IN MAIN PROGRAM BODY
// =================================================================
fbBlinkTimer(IN := NOT fbBlinkTimer.Q, PT := T#500MS);

IF fbBlinkTimer.Q AND NOT bBlinkTimer_Q_Old THEN
	GVL_MASTER.bBlink_1Hz := NOT GVL_MASTER.bBlink_1Hz;
END_IF
bBlinkTimer_Q_Old := fbBlinkTimer.Q;

// =================================================================
// REFRESH LOCAL SYSTEM TIME & FORMAT STRINGS (O que faltava aqui!)
// =================================================================
fbLocalTime(bEnable := TRUE); // Executa o bloco para ler a hora do Windows

IF fbLocalTime.bValid THEN
	
	// --- FORMATAÇÃO DA HORA (sTimeReal) ---
	IF fbLocalTime.systemTime.wHour < 10 THEN
		sTimeReal := CONCAT('0', WORD_TO_STRING(fbLocalTime.systemTime.wHour));
	ELSE
		sTimeReal := WORD_TO_STRING(fbLocalTime.systemTime.wHour);
	END_IF
	
	sTimeReal := CONCAT(sTimeReal, ':');
	
	IF fbLocalTime.systemTime.wMinute < 10 THEN
		sTimeReal := CONCAT(sTimeReal, CONCAT('0', WORD_TO_STRING(fbLocalTime.systemTime.wMinute)));
	ELSE
		sTimeReal := CONCAT(sTimeReal, WORD_TO_STRING(fbLocalTime.systemTime.wMinute));
	END_IF
	
	// --- FORMATAÇÃO DA DATA (sCurrentTimeStr) ---
	IF fbLocalTime.systemTime.wDay < 10 THEN
		sCurrentTimeStr := CONCAT('0', WORD_TO_STRING(fbLocalTime.systemTime.wDay));
	ELSE
		sCurrentTimeStr := WORD_TO_STRING(fbLocalTime.systemTime.wDay);
	END_IF
	
	sCurrentTimeStr := CONCAT(sCurrentTimeStr, '/');
	
	IF fbLocalTime.systemTime.wMonth < 10 THEN
		sCurrentTimeStr := CONCAT(sCurrentTimeStr, CONCAT('0', WORD_TO_STRING(fbLocalTime.systemTime.wMonth)));
	ELSE
		sCurrentTimeStr := CONCAT(sCurrentTimeStr, WORD_TO_STRING(fbLocalTime.systemTime.wMonth));
	END_IF
	
	sCurrentTimeStr := CONCAT(sCurrentTimeStr, '/');
	sCurrentTimeStr := CONCAT(sCurrentTimeStr, WORD_TO_STRING(fbLocalTime.systemTime.wYear));

END_IF

// =================================================================
// ALARM TRIGGER TEST BLOCK (EDGE DETECTION)
// =================================================================
fbTestAlarmTrigger(CLK := bTriggerTestAlarm);

IF fbTestAlarmTrigger.Q THEN
	// Agora as strings sTimeReal e sCurrentTimeStr já possuem valor real!
	M_AddLogToHistory(
		sTime		:= sTimeReal,
		sType 		:= E_Alarms.FAULT,
		sDate		:= sCurrentTimeStr, 
		abType		:= E_Alarms.FAULT,
		nEventId	:= 3001,
		sMessage	:= 'Error feio'
	);
		M_AddLogToHistory(
		sTime		:= sTimeReal,
		sType 		:= E_Alarms.Cycle_Stop_Fault,
		sDate		:= sCurrentTimeStr, 
		abType		:= E_Alarms.FAULT,
		nEventId	:= 3001,
		sMessage	:= 'Error feio'
	);
		M_AddLogToHistory(
		sTime		:= sTimeReal,
		sType 		:= E_Alarms.Cycle_Stop_Request,
		sDate		:= sCurrentTimeStr, 
		abType		:= 2,
		nEventId	:= 3001,
		sMessage	:= 'Error feio'
		
		);
		M_AddLogToHistory(
		sTime		:= sTimeReal,
		sType 		:= E_Alarms.MESSAGE,
		sDate		:= sCurrentTimeStr, 
		abType		:= 3,
		nEventId	:= 3001,
		sMessage	:= 'Error feio'
	);
END_IF

// =================================================================
// NOW CALL THE METHOD TO PROCESS STRINGS AND HMI COLORS
// =================================================================
M_StatusHMI();
M_PLC_Power();

METHOD M_AddLogToHistory
VAR_INPUT
	sTime		: STRING(255);
	sType		: E_Alarms;
	sDate		: STRING(255);
	abType		: DINT;	
	nEventId	: INT;
	sMessage	: STRING(255);
END_VAR
VAR
	i           : INT; // Loop index variable for shifting
END_VAR
// 1. Cascade existing array rows downward to create an empty slot at index [1]
FOR i := 100 TO 2 BY -1 DO
	GVL_HMI.arrAlarmHistory[i] := GVL_HMI.arrAlarmHistory[i - 1];
END_FOR

// 2. Inject the newest event block directly into the primary top row
GVL_HMI.arrAlarmHistory[1].sTime     := sTime;
GVL_HMI.arrAlarmHistory[1].sType     := sType;
GVL_HMI.arrAlarmHistory[1].sDate     := sDate;
GVL_HMI.arrAlarmHistory[1].abType    := abType;
GVL_HMI.arrAlarmHistory[1].nEventId  := nEventId;
GVL_HMI.arrAlarmHistory[1].sMessage  := sMessage;
// 
// // 3. Drive high-priority alert strings and colors onto the main overhead header banner
// IF eSeverity >= E_Alarms.ERROR THEN
// 	GVL_HMI.StatusHMI.sMachineStatusText := sMessage;      // Texto central do Banner
// 	GVL_HMI.StatusHMI.sBannerBckColor   := '#FF0000';     // Fundo Vermelho para Erros/Críticos
// 	GVL_HMI.StatusHMI.sBannerTextColor   := '#FFFFFF';     // Texto Branco para dar contraste
// ELSIF eSeverity = E_Alarms.WARNING THEN
// 	GVL_HMI.StatusHMI.sMachineStatusText := sMessage;
// 	GVL_HMI.StatusHMI.sBannerBckColor   := '#FF8C00';     // Fundo Laranja para Avisos
// 	GVL_HMI.StatusHMI.sBannerTextColor   := '#FFFFFF';
// END_IF
END_METHOD

METHOD M_PLC_Power
VAR_INPUT
END_VAR
// =========================================================================
// 1. TIMER CONFIGURATION (Dynamic PT based on Command)
// =========================================================================
// Define the preset time (PT) dynamically depending on the selected action
IF GVL_HMI.ePowerCmd = E_PLC_Power.Reboot THEN
    tonPowerDelay.PT := T#15S;
ELSIF GVL_HMI.ePowerCmd = E_PLC_Power.Shutdown THEN
    tonPowerDelay.PT := T#60S;
END_IF

// Call the timer block first so it updates its Elapsed Time (.ET)
tonPowerDelay(
    IN := (GVL_HMI.ePowerCmd = E_PLC_Power.Reboot OR GVL_HMI.ePowerCmd = E_PLC_Power.Shutdown)
);

// Calculate countdown value for HMI visualization after the timer execution
IF tonPowerDelay.IN THEN
    IF GVL_HMI.ePowerCmd = E_PLC_Power.Shutdown THEN
        iCountdownValue := DINT_TO_INT(60 - (TIME_TO_DINT(tonPowerDelay.ET) / 1000));
    ELSIF GVL_HMI.ePowerCmd = E_PLC_Power.Reboot THEN
        iCountdownValue := DINT_TO_INT(15 - (TIME_TO_DINT(tonPowerDelay.ET) / 1000));
    END_IF
ELSE 
    iCountdownValue := 60; // Default state idle value
END_IF
// =========================================================================
// 2. STATE MACHINE WITH CANCEL FUNCTIONALITY
// =========================================================================
CASE GVL_HMI.ePowerCmd OF
    
    E_PLC_Power.Idle:
        bTriggerReboot   := FALSE;
        bTriggerShutdown := FALSE;

    E_PLC_Power.Reboot:
        // Triggers the reboot block ONLY after the 60 seconds expire
        IF tonPowerDelay.Q THEN
            bTriggerReboot := TRUE;
        END_IF

    E_PLC_Power.Shutdown:
        // Triggers the shutdown block ONLY after the 60 seconds expire
        IF tonPowerDelay.Q THEN
            bTriggerShutdown := TRUE;
        END_IF
// 	E_PLC_Power.ExitHMI:
//             bTriggerExitHMI := TRUE;


    E_PLC_Power.Cancel:
        // Safe abortion: clears all triggers and forces state back to Idle immediately
        bTriggerReboot    := FALSE;
        bTriggerShutdown  := FALSE;
        GVL_HMI.ePowerCmd := E_PLC_Power.Idle;

END_CASE

// =========================================================================
// 3. HARDWARE & OS BLOCK EXECUTION (ADS COMMANDS)
// =========================================================================
fbReboot(
    NETID := '',
    START := bTriggerReboot,
    TMOUT := DEFAULT_ADS_TIMEOUT
);

fbShutdown(
    NETID := '',
    START := bTriggerShutdown,
    TMOUT := DEFAULT_ADS_TIMEOUT
);

// fbKillEdge(
//     NETID:= '',
//     PATHSTR:= 'C:\Windows\System32\taskkill.exe',
//     COMNDLINE:= '/F /IM msedge.exe /T', // <--- Corrigido para msedge.exe com "e"
//     START:= (GVL_HMI.ePowerCmd = E_PLC_Power.ExitHMI),
//     TMOUT:= DEFAULT_ADS_TIMEOUT
// );
// =========================================================================
// 4. CLEAN & SAFE RESET
// =========================================================================
IF fbReboot.BUSY OR fbReboot.ERR THEN
    bTriggerReboot    := FALSE;
    GVL_HMI.ePowerCmd := E_PLC_Power.Idle;
END_IF

IF fbShutdown.BUSY OR fbShutdown.ERR THEN
    bTriggerShutdown  := FALSE;
    GVL_HMI.ePowerCmd := E_PLC_Power.Idle;
END_IF

// IF fbKillEdge.BUSY OR fbKillEdge.ERR THEN
// 	bTriggerExitHMI  := FALSE;
//     GVL_HMI.ePowerCmd := E_PLC_Power.Idle;
// END_IF
END_METHOD

METHOD M_StatusHMI : BOOL
VAR
// sGreen				:STRING := '{"color":"rgba(0, 180, 0, 1)"}';	
// sREd				:STRING := '{"color":"rgba(255, 0, 0, 1)"}';    
// sWhite				:STRING := '{"color":"rgba(255, 255, 255, 1)"}';
// sBlack				:STRING := '{"color":"rgba(0, 0, 0, 1)"}';
// sGrey				:STRING := '{"color":"rgba(128, 128, 128, 1)"}';
// sYellow				:STRING := '{"color":"rgba(255, 255, 0, 1)"}';
// sTransparent		:STRING := '{"color":"rgba(0, 0, 0, 0)"}'; 

END_VAR

bFlash := GVL_MASTER.bBlink_1Hz;



CASE GVL_MASTER.stMachineStatus.eMachineState OF

    E_MachineState.SYSTEM_INITIALISING:
        GVL_HMI.StatusHMI.sMachineStatusText := 'SYSTEM INITIALIZING';        
        GVL_HMI.StatusHMI.sBannerBckColor    := GVL_HMI.sYELLOW; 
        GVL_HMI.StatusHMI.sBannerTextColor   := GVL_HMI.sBLACK;

    E_MachineState.SYSTEM_READY_TO_START:
        GVL_HMI.StatusHMI.sMachineStatusText := 'SYSTEM READY TO START';        
        IF bFlash THEN
            GVL_HMI.StatusHMI.sBannerBckColor  := GVL_HMI.sGREEN;
            GVL_HMI.StatusHMI.sBannerTextColor := GVL_HMI.sWHITE;
        ELSE    
            GVL_HMI.StatusHMI.sBannerBckColor  := GVL_HMI.sWHITE;
            GVL_HMI.StatusHMI.sBannerTextColor := GVL_HMI.sGREEN;
        END_IF

    E_MachineState.SYSTEM_AUTO_CYCLE:
        GVL_HMI.StatusHMI.sMachineStatusText := 'SYSTEM AUTO CYCLE';        
        GVL_HMI.StatusHMI.sBannerBckColor    := GVL_HMI.sGREEN;
        GVL_HMI.StatusHMI.sBannerTextColor   := GVL_HMI.sWHITE; 

    E_MachineState.STOPPING:
        GVL_HMI.StatusHMI.sMachineStatusText := 'STOPPING';        
        IF bFlash THEN    
            GVL_HMI.StatusHMI.sBannerBckColor  := GVL_HMI.sGREY;
            GVL_HMI.StatusHMI.sBannerTextColor := GVL_HMI.sWHITE;    
        ELSE    
            GVL_HMI.StatusHMI.sBannerBckColor  := GVL_HMI.sTRANSP;
            GVL_HMI.StatusHMI.sBannerTextColor := GVL_HMI.sBLACK;     
        END_IF

    E_MachineState.STOPPED:
        GVL_HMI.StatusHMI.sMachineStatusText := 'CYCLE STOPPED';        
        GVL_HMI.StatusHMI.sBannerBckColor    := GVL_HMI.sGREY;
        GVL_HMI.StatusHMI.sBannerTextColor   := GVL_HMI.sWHITE;    

    E_MachineState.FAULT:
        GVL_HMI.StatusHMI.sMachineStatusText := 'IMMEDIATE FAULT';        
        IF bFlash THEN    
            GVL_HMI.StatusHMI.sBannerBckColor  := GVL_HMI.sREDFail;
            GVL_HMI.StatusHMI.sBannerTextColor := GVL_HMI.sWHITE;   
        ELSE    
            GVL_HMI.StatusHMI.sBannerBckColor  := GVL_HMI.sWHITE;
            GVL_HMI.StatusHMI.sBannerTextColor := GVL_HMI.sREDFail;
        END_IF
	E_MachineState.MANUAL_MODE:
        GVL_HMI.StatusHMI.sMachineStatusText := 'MANUAL MODE';        
        GVL_HMI.StatusHMI.sBannerBckColor  := GVL_HMI.sBLUEInProgress;
        GVL_HMI.StatusHMI.sBannerTextColor := GVL_HMI.sWHITE;   


END_CASE


M_StatusHMI := TRUE;
END_METHOD

END_PROGRAM
